REGION Network 3: Vaciado
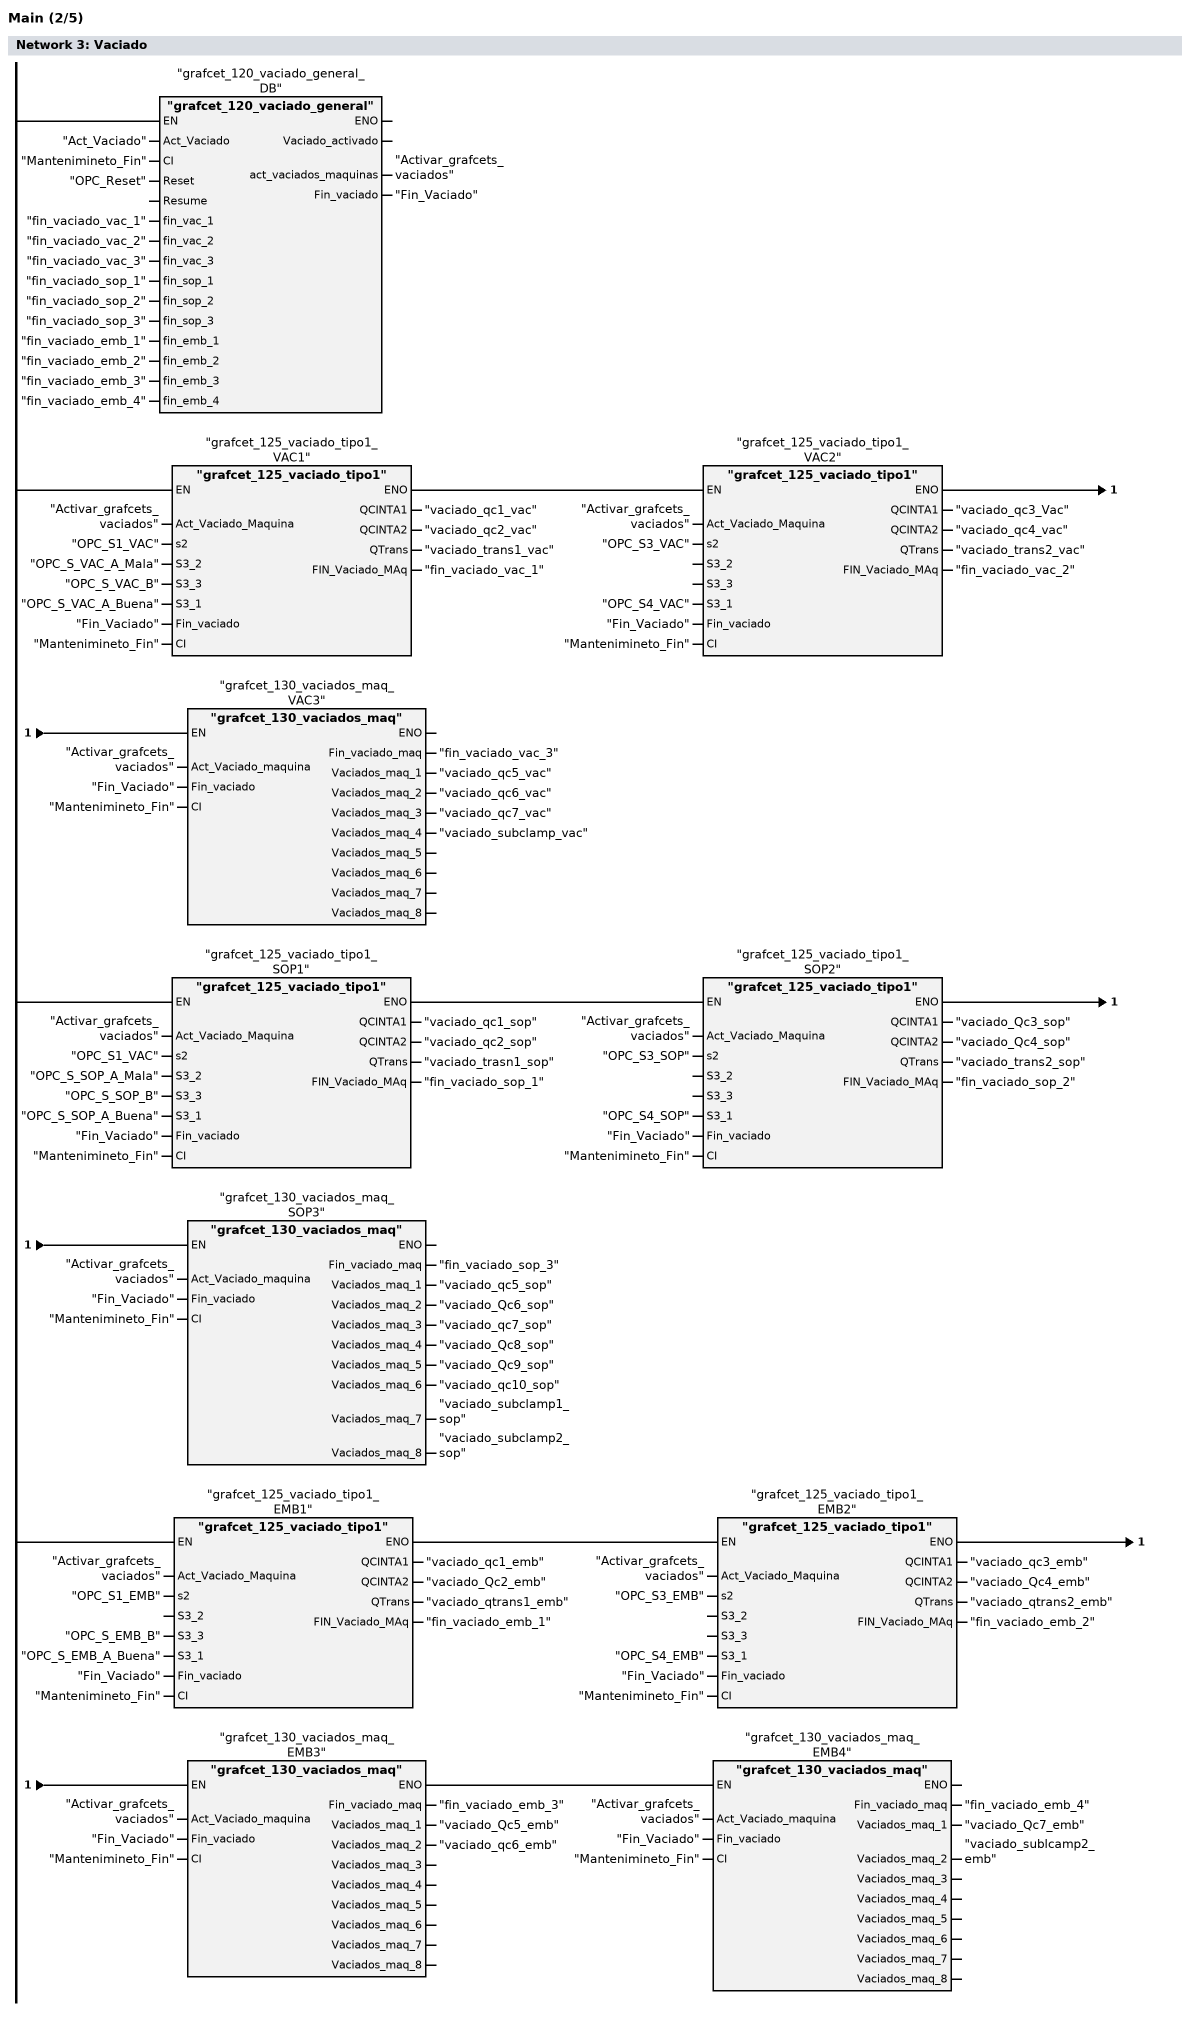
   RUNG wire#powerrail
      "grafcet_120_vaciado_general_DB"(Act_Vaciado := "Act_Vaciado", CI := "Mantenimineto_Fin", Reset := "OPC_Reset", Resume :=, fin_vac_1 := "fin_vaciado_vac_1", fin_vac_2 := "fin_vaciado_vac_2", fin_vac_3 := "fin_vaciado_vac_3", fin_sop_1 := "fin_vaciado_sop_1", fin_sop_2 := "fin_vaciado_sop_2", fin_sop_3 := "fin_vaciado_sop_3", fin_emb_1 := "fin_vaciado_emb_1", fin_emb_2 := "fin_vaciado_emb_2", fin_emb_3 := "fin_vaciado_emb_3", fin_emb_4 := "fin_vaciado_emb_4", Vaciado_activado =>, act_vaciados_maquinas => "Activar_grafcets_vaciados", Fin_vaciado => "Fin_Vaciado")
   END_RUNG
   RUNG wire#powerrail
      "grafcet_125_vaciado_tipo1_VAC1"(Act_Vaciado_Maquina := "Activar_grafcets_vaciados", s2 := "OPC_S1_VAC", S3_2 := "OPC_S_VAC_A_Mala", S3_3 := "OPC_S_VAC_B", S3_1 := "OPC_S_VAC_A_Buena", Fin_vaciado := "Fin_Vaciado", CI := "Mantenimineto_Fin", QCINTA1 => "vaciado_qc1_vac", QCINTA2 => "vaciado_qc2_vac", QTrans => "vaciado_trans1_vac", FIN_Vaciado_MAq => "fin_vaciado_vac_1")
      "grafcet_125_vaciado_tipo1_VAC2"(Act_Vaciado_Maquina := "Activar_grafcets_vaciados", s2 := "OPC_S3_VAC", S3_2 :=, S3_3 :=, S3_1 := "OPC_S4_VAC", Fin_vaciado := "Fin_Vaciado", CI := "Mantenimineto_Fin", QCINTA1 => "vaciado_qc3_Vac", QCINTA2 => "vaciado_qc4_vac", QTrans => "vaciado_trans2_vac", FIN_Vaciado_MAq => "fin_vaciado_vac_2")
      "grafcet_130_vaciados_maq_VAC3"(Act_Vaciado_maquina := "Activar_grafcets_vaciados", Fin_vaciado := "Fin_Vaciado", CI := "Mantenimineto_Fin", Fin_vaciado_maq => "fin_vaciado_vac_3", Vaciados_maq_1 => "vaciado_qc5_vac", Vaciados_maq_2 => "vaciado_qc6_vac", Vaciados_maq_3 => "vaciado_qc7_vac", Vaciados_maq_4 => "vaciado_subclamp_vac", Vaciados_maq_5 =>, Vaciados_maq_6 =>, Vaciados_maq_7 =>, Vaciados_maq_8 =>)
   END_RUNG
   RUNG wire#powerrail
      "grafcet_125_vaciado_tipo1_SOP1"(Act_Vaciado_Maquina := "Activar_grafcets_vaciados", s2 := "OPC_S1_VAC", S3_2 := "OPC_S_SOP_A_Mala", S3_3 := "OPC_S_SOP_B", S3_1 := "OPC_S_SOP_A_Buena", Fin_vaciado := "Fin_Vaciado", CI := "Mantenimineto_Fin", QCINTA1 => "vaciado_qc1_sop", QCINTA2 => "vaciado_qc2_sop", QTrans => "vaciado_trasn1_sop", FIN_Vaciado_MAq => "fin_vaciado_sop_1")
      "grafcet_125_vaciado_tipo1_SOP2"(Act_Vaciado_Maquina := "Activar_grafcets_vaciados", s2 := "OPC_S3_SOP", S3_2 :=, S3_3 :=, S3_1 := "OPC_S4_SOP", Fin_vaciado := "Fin_Vaciado", CI := "Mantenimineto_Fin", QCINTA1 => "vaciado_Qc3_sop", QCINTA2 => "vaciado_Qc4_sop", QTrans => "vaciado_trans2_sop", FIN_Vaciado_MAq => "fin_vaciado_sop_2")
      "grafcet_130_vaciados_maq_SOP3"(Act_Vaciado_maquina := "Activar_grafcets_vaciados", Fin_vaciado := "Fin_Vaciado", CI := "Mantenimineto_Fin", Fin_vaciado_maq => "fin_vaciado_sop_3", Vaciados_maq_1 => "vaciado_qc5_sop", Vaciados_maq_2 => "vaciado_Qc6_sop", Vaciados_maq_3 => "vaciado_qc7_sop", Vaciados_maq_4 => "vaciado_Qc8_sop", Vaciados_maq_5 => "vaciado_Qc9_sop", Vaciados_maq_6 => "vaciado_qc10_sop", Vaciados_maq_7 => "vaciado_subclamp1_sop", Vaciados_maq_8 => "vaciado_subclamp2_sop")
   END_RUNG
   RUNG wire#powerrail
      "grafcet_125_vaciado_tipo1_EMB1"(Act_Vaciado_Maquina := "Activar_grafcets_vaciados", s2 := "OPC_S1_EMB", S3_2 :=, S3_3 := "OPC_S_EMB_B", S3_1 := "OPC_S_EMB_A_Buena", Fin_vaciado := "Fin_Vaciado", CI := "Mantenimineto_Fin", QCINTA1 => "vaciado_qc1_emb", QCINTA2 => "vaciado_Qc2_emb", QTrans => "vaciado_qtrans1_emb", FIN_Vaciado_MAq => "fin_vaciado_emb_1")
      "grafcet_125_vaciado_tipo1_EMB2"(Act_Vaciado_Maquina := "Activar_grafcets_vaciados", s2 := "OPC_S3_EMB", S3_2 :=, S3_3 :=, S3_1 := "OPC_S4_EMB", Fin_vaciado := "Fin_Vaciado", CI := "Mantenimineto_Fin", QCINTA1 => "vaciado_qc3_emb", QCINTA2 => "vaciado_Qc4_emb", QTrans => "vaciado_qtrans2_emb", FIN_Vaciado_MAq => "fin_vaciado_emb_2")
      "grafcet_130_vaciados_maq_EMB3"(Act_Vaciado_maquina := "Activar_grafcets_vaciados", Fin_vaciado := "Fin_Vaciado", CI := "Mantenimineto_Fin", Fin_vaciado_maq => "fin_vaciado_emb_3", Vaciados_maq_1 => "vaciado_Qc5_emb", Vaciados_maq_2 => "vaciado_qc6_emb", Vaciados_maq_3 =>, Vaciados_maq_4 =>, Vaciados_maq_5 =>, Vaciados_maq_6 =>, Vaciados_maq_7 =>, Vaciados_maq_8 =>)
      "grafcet_130_vaciados_maq_EMB4"(Act_Vaciado_maquina := "Activar_grafcets_vaciados", Fin_vaciado := "Fin_Vaciado", CI := "Mantenimineto_Fin", Fin_vaciado_maq => "fin_vaciado_emb_4", Vaciados_maq_1 => "vaciado_Qc7_emb", Vaciados_maq_2 => "vaciado_sublcamp2_emb", Vaciados_maq_3 =>, Vaciados_maq_4 =>, Vaciados_maq_5 =>, Vaciados_maq_6 =>, Vaciados_maq_7 =>, Vaciados_maq_8 =>)
   END_RUNG
   // the same network as SCL:
   "grafcet_120_vaciado_general_DB"(Act_Vaciado := "Act_Vaciado",   // "grafcet_120_vaciado_general"
                           CI := "Mantenimineto_Fin",
                           Reset := "OPC_Reset",
                           fin_vac_1 := "fin_vaciado_vac_1",
                           fin_vac_2 := "fin_vaciado_vac_2",
                           fin_vac_3 := "fin_vaciado_vac_3",
                           fin_sop_1 := "fin_vaciado_sop_1",
                           fin_sop_2 := "fin_vaciado_sop_2",
                           fin_sop_3 := "fin_vaciado_sop_3",
                           fin_emb_1 := "fin_vaciado_emb_1",
                           fin_emb_2 := "fin_vaciado_emb_2",
                           fin_emb_3 := "fin_vaciado_emb_3",
                           fin_emb_4 := "fin_vaciado_emb_4",
                           act_vaciados_maquinas => "Activar_grafcets_vaciados",
                           Fin_vaciado => "Fin_Vaciado");
   "grafcet_125_vaciado_tipo1_VAC1"(Act_Vaciado_Maquina := "Activar_grafcets_vaciados",   // "grafcet_125_vaciado_tipo1"
                           s2 := "OPC_S1_VAC",
                           S3_2 := "OPC_S_VAC_A_Mala",
                           S3_3 := "OPC_S_VAC_B",
                           S3_1 := "OPC_S_VAC_A_Buena",
                           Fin_vaciado := "Fin_Vaciado",
                           CI := "Mantenimineto_Fin",
                           QCINTA1 => "vaciado_qc1_vac",
                           QCINTA2 => "vaciado_qc2_vac",
                           QTrans => "vaciado_trans1_vac",
                           FIN_Vaciado_MAq => "fin_vaciado_vac_1",
                           ENO => #_w1);
   "grafcet_125_vaciado_tipo1_VAC2"(EN := #_w1,   // "grafcet_125_vaciado_tipo1"
                           Act_Vaciado_Maquina := "Activar_grafcets_vaciados",
                           s2 := "OPC_S3_VAC",
                           S3_1 := "OPC_S4_VAC",
                           Fin_vaciado := "Fin_Vaciado",
                           CI := "Mantenimineto_Fin",
                           QCINTA1 => "vaciado_qc3_Vac",
                           QCINTA2 => "vaciado_qc4_vac",
                           QTrans => "vaciado_trans2_vac",
                           FIN_Vaciado_MAq => "fin_vaciado_vac_2",
                           ENO => #_w2);
   IF #_w2 THEN
       "grafcet_130_vaciados_maq_VAC3"(Act_Vaciado_maquina := "Activar_grafcets_vaciados",   // "grafcet_130_vaciados_maq"
                               Fin_vaciado := "Fin_Vaciado",
                               CI := "Mantenimineto_Fin",
                               Fin_vaciado_maq => "fin_vaciado_vac_3",
                               Vaciados_maq_1 => "vaciado_qc5_vac",
                               Vaciados_maq_2 => "vaciado_qc6_vac",
                               Vaciados_maq_3 => "vaciado_qc7_vac",
                               Vaciados_maq_4 => "vaciado_subclamp_vac");
   END_IF;
   "grafcet_125_vaciado_tipo1_SOP1"(Act_Vaciado_Maquina := "Activar_grafcets_vaciados",   // "grafcet_125_vaciado_tipo1"
                           s2 := "OPC_S1_VAC",
                           S3_2 := "OPC_S_SOP_A_Mala",
                           S3_3 := "OPC_S_SOP_B",
                           S3_1 := "OPC_S_SOP_A_Buena",
                           Fin_vaciado := "Fin_Vaciado",
                           CI := "Mantenimineto_Fin",
                           QCINTA1 => "vaciado_qc1_sop",
                           QCINTA2 => "vaciado_qc2_sop",
                           QTrans => "vaciado_trasn1_sop",
                           FIN_Vaciado_MAq => "fin_vaciado_sop_1",
                           ENO => #_w3);
   "grafcet_125_vaciado_tipo1_SOP2"(EN := #_w3,   // "grafcet_125_vaciado_tipo1"
                           Act_Vaciado_Maquina := "Activar_grafcets_vaciados",
                           s2 := "OPC_S3_SOP",
                           S3_1 := "OPC_S4_SOP",
                           Fin_vaciado := "Fin_Vaciado",
                           CI := "Mantenimineto_Fin",
                           QCINTA1 => "vaciado_Qc3_sop",
                           QCINTA2 => "vaciado_Qc4_sop",
                           QTrans => "vaciado_trans2_sop",
                           FIN_Vaciado_MAq => "fin_vaciado_sop_2",
                           ENO => #_w4);
   IF #_w4 THEN
       "grafcet_130_vaciados_maq_SOP3"(Act_Vaciado_maquina := "Activar_grafcets_vaciados",   // "grafcet_130_vaciados_maq"
                               Fin_vaciado := "Fin_Vaciado",
                               CI := "Mantenimineto_Fin",
                               Fin_vaciado_maq => "fin_vaciado_sop_3",
                               Vaciados_maq_1 => "vaciado_qc5_sop",
                               Vaciados_maq_2 => "vaciado_Qc6_sop",
                               Vaciados_maq_3 => "vaciado_qc7_sop",
                               Vaciados_maq_4 => "vaciado_Qc8_sop",
                               Vaciados_maq_5 => "vaciado_Qc9_sop",
                               Vaciados_maq_6 => "vaciado_qc10_sop",
                               Vaciados_maq_7 => "vaciado_subclamp1_sop",
                               Vaciados_maq_8 => "vaciado_subclamp2_sop");
   END_IF;
   "grafcet_125_vaciado_tipo1_EMB1"(Act_Vaciado_Maquina := "Activar_grafcets_vaciados",   // "grafcet_125_vaciado_tipo1"
                           s2 := "OPC_S1_EMB",
                           S3_3 := "OPC_S_EMB_B",
                           S3_1 := "OPC_S_EMB_A_Buena",
                           Fin_vaciado := "Fin_Vaciado",
                           CI := "Mantenimineto_Fin",
                           QCINTA1 => "vaciado_qc1_emb",
                           QCINTA2 => "vaciado_Qc2_emb",
                           QTrans => "vaciado_qtrans1_emb",
                           FIN_Vaciado_MAq => "fin_vaciado_emb_1",
                           ENO => #_w5);
   "grafcet_125_vaciado_tipo1_EMB2"(EN := #_w5,   // "grafcet_125_vaciado_tipo1"
                           Act_Vaciado_Maquina := "Activar_grafcets_vaciados",
                           s2 := "OPC_S3_EMB",
                           S3_1 := "OPC_S4_EMB",
                           Fin_vaciado := "Fin_Vaciado",
                           CI := "Mantenimineto_Fin",
                           QCINTA1 => "vaciado_qc3_emb",
                           QCINTA2 => "vaciado_Qc4_emb",
                           QTrans => "vaciado_qtrans2_emb",
                           FIN_Vaciado_MAq => "fin_vaciado_emb_2",
                           ENO => #_w6);
   "grafcet_130_vaciados_maq_EMB3"(EN := #_w6,   // "grafcet_130_vaciados_maq"
                           Act_Vaciado_maquina := "Activar_grafcets_vaciados",
                           Fin_vaciado := "Fin_Vaciado",
                           CI := "Mantenimineto_Fin",
                           Fin_vaciado_maq => "fin_vaciado_emb_3",
                           Vaciados_maq_1 => "vaciado_Qc5_emb",
                           Vaciados_maq_2 => "vaciado_qc6_emb",
                           ENO => #_w7);
   IF #_w7 THEN
       "grafcet_130_vaciados_maq_EMB4"(Act_Vaciado_maquina := "Activar_grafcets_vaciados",   // "grafcet_130_vaciados_maq"
                               Fin_vaciado := "Fin_Vaciado",
                               CI := "Mantenimineto_Fin",
                               Fin_vaciado_maq => "fin_vaciado_emb_4",
                               Vaciados_maq_1 => "vaciado_Qc7_emb",
                               Vaciados_maq_2 => "vaciado_sublcamp2_emb");
   END_IF;
END_REGION

REGION Network 4: Maquina Vacunas
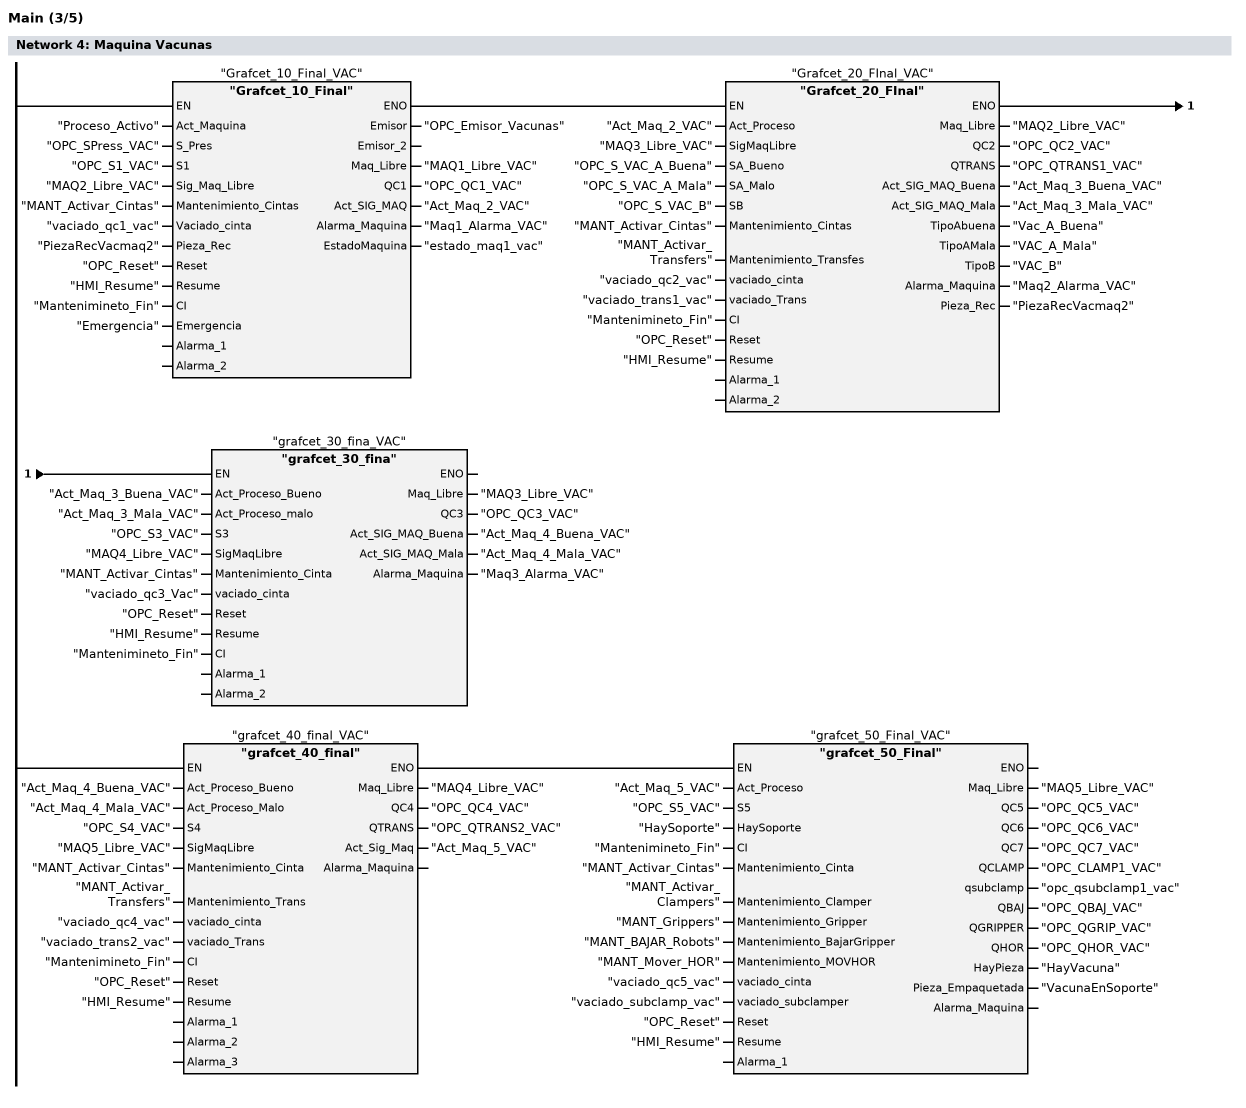
   RUNG wire#powerrail
      "Grafcet_10_Final_VAC"(Act_Maquina := "Proceso_Activo", S_Pres := "OPC_SPress_VAC", S1 := "OPC_S1_VAC", Sig_Maq_Libre := "MAQ2_Libre_VAC", Mantenimiento_Cintas := "MANT_Activar_Cintas", Vaciado_cinta := "vaciado_qc1_vac", Pieza_Rec := "PiezaRecVacmaq2", Reset := "OPC_Reset", Resume := "HMI_Resume", CI := "Mantenimineto_Fin", Emergencia := "Emergencia", Alarma_1 :=, Alarma_2 :=, Emisor => "OPC_Emisor_Vacunas", Emisor_2 =>, Maq_Libre => "MAQ1_Libre_VAC", QC1 => "OPC_QC1_VAC", Act_SIG_MAQ => "Act_Maq_2_VAC", Alarma_Maquina => "Maq1_Alarma_VAC", EstadoMaquina => "estado_maq1_vac")
      "Grafcet_20_FInal_VAC"(Act_Proceso := "Act_Maq_2_VAC", SigMaqLibre := "MAQ3_Libre_VAC", SA_Bueno := "OPC_S_VAC_A_Buena", SA_Malo := "OPC_S_VAC_A_Mala", SB := "OPC_S_VAC_B", Mantenimiento_Cintas := "MANT_Activar_Cintas", Mantenimiento_Transfes := "MANT_Activar_Transfers", vaciado_cinta := "vaciado_qc2_vac", vaciado_Trans := "vaciado_trans1_vac", CI := "Mantenimineto_Fin", Reset := "OPC_Reset", Resume := "HMI_Resume", Alarma_1 :=, Alarma_2 :=, Maq_Libre => "MAQ2_Libre_VAC", QC2 => "OPC_QC2_VAC", QTRANS => "OPC_QTRANS1_VAC", Act_SIG_MAQ_Buena => "Act_Maq_3_Buena_VAC", Act_SIG_MAQ_Mala => "Act_Maq_3_Mala_VAC", TipoAbuena => "Vac_A_Buena", TipoAMala => "VAC_A_Mala", TipoB => "VAC_B", Alarma_Maquina => "Maq2_Alarma_VAC", Pieza_Rec => "PiezaRecVacmaq2")
      "grafcet_30_fina_VAC"(Act_Proceso_Bueno := "Act_Maq_3_Buena_VAC", Act_Proceso_malo := "Act_Maq_3_Mala_VAC", S3 := "OPC_S3_VAC", SigMaqLibre := "MAQ4_Libre_VAC", Mantenimiento_Cinta := "MANT_Activar_Cintas", vaciado_cinta := "vaciado_qc3_Vac", Reset := "OPC_Reset", Resume := "HMI_Resume", CI := "Mantenimineto_Fin", Alarma_1 :=, Alarma_2 :=, Maq_Libre => "MAQ3_Libre_VAC", QC3 => "OPC_QC3_VAC", Act_SIG_MAQ_Buena => "Act_Maq_4_Buena_VAC", Act_SIG_MAQ_Mala => "Act_Maq_4_Mala_VAC", Alarma_Maquina => "Maq3_Alarma_VAC")
   END_RUNG
   RUNG wire#powerrail
      "grafcet_40_final_VAC"(Act_Proceso_Bueno := "Act_Maq_4_Buena_VAC", Act_Proceso_Malo := "Act_Maq_4_Mala_VAC", S4 := "OPC_S4_VAC", SigMaqLibre := "MAQ5_Libre_VAC", Mantenimiento_Cinta := "MANT_Activar_Cintas", Mantenimiento_Trans := "MANT_Activar_Transfers", vaciado_cinta := "vaciado_qc4_vac", vaciado_Trans := "vaciado_trans2_vac", CI := "Mantenimineto_Fin", Reset := "OPC_Reset", Resume := "HMI_Resume", Alarma_1 :=, Alarma_2 :=, Alarma_3 :=, Maq_Libre => "MAQ4_Libre_VAC", QC4 => "OPC_QC4_VAC", QTRANS => "OPC_QTRANS2_VAC", Act_Sig_Maq => "Act_Maq_5_VAC", Alarma_Maquina =>)
      "grafcet_50_Final_VAC"(Act_Proceso := "Act_Maq_5_VAC", S5 := "OPC_S5_VAC", HaySoporte := "HaySoporte", CI := "Mantenimineto_Fin", Mantenimiento_Cinta := "MANT_Activar_Cintas", Mantenimiento_Clamper := "MANT_Activar_Clampers", Mantenimiento_Gripper := "MANT_Grippers", Mantenimiento_BajarGripper := "MANT_BAJAR_Robots", Mantenimiento_MOVHOR := "MANT_Mover_HOR", vaciado_cinta := "vaciado_qc5_vac", vaciado_subclamper := "vaciado_subclamp_vac", Reset := "OPC_Reset", Resume := "HMI_Resume", Alarma_1 :=, Maq_Libre => "MAQ5_Libre_VAC", QC5 => "OPC_QC5_VAC", QC6 => "OPC_QC6_VAC", QC7 => "OPC_QC7_VAC", QCLAMP => "OPC_CLAMP1_VAC", qsubclamp => "opc_qsubclamp1_vac", QBAJ => "OPC_QBAJ_VAC", QGRIPPER => "OPC_QGRIP_VAC", QHOR => "OPC_QHOR_VAC", HayPieza => "HayVacuna", Pieza_Empaquetada => "VacunaEnSoporte", Alarma_Maquina =>)
   END_RUNG
   // the same network as SCL:
   "Grafcet_10_Final_VAC"(Act_Maquina := "Proceso_Activo",   // "Grafcet_10_Final"
                          S_Pres := "OPC_SPress_VAC",
                          S1 := "OPC_S1_VAC",
                          Sig_Maq_Libre := "MAQ2_Libre_VAC",
                          Mantenimiento_Cintas := "MANT_Activar_Cintas",
                          Vaciado_cinta := "vaciado_qc1_vac",
                          Pieza_Rec := "PiezaRecVacmaq2",
                          Reset := "OPC_Reset",
                          Resume := "HMI_Resume",
                          CI := "Mantenimineto_Fin",
                          Emergencia := "Emergencia",
                          Emisor => "OPC_Emisor_Vacunas",
                          Maq_Libre => "MAQ1_Libre_VAC",
                          QC1 => "OPC_QC1_VAC",
                          Act_SIG_MAQ => "Act_Maq_2_VAC",
                          Alarma_Maquina => "Maq1_Alarma_VAC",
                          EstadoMaquina => "estado_maq1_vac",
                          ENO => #_w1);
   "Grafcet_20_FInal_VAC"(EN := #_w1,   // "Grafcet_20_FInal"
                          Act_Proceso := "Act_Maq_2_VAC",
                          SigMaqLibre := "MAQ3_Libre_VAC",
                          SA_Bueno := "OPC_S_VAC_A_Buena",
                          SA_Malo := "OPC_S_VAC_A_Mala",
                          SB := "OPC_S_VAC_B",
                          Mantenimiento_Cintas := "MANT_Activar_Cintas",
                          Mantenimiento_Transfes := "MANT_Activar_Transfers",
                          vaciado_cinta := "vaciado_qc2_vac",
                          vaciado_Trans := "vaciado_trans1_vac",
                          CI := "Mantenimineto_Fin",
                          Reset := "OPC_Reset",
                          Resume := "HMI_Resume",
                          Maq_Libre => "MAQ2_Libre_VAC",
                          QC2 => "OPC_QC2_VAC",
                          QTRANS => "OPC_QTRANS1_VAC",
                          Act_SIG_MAQ_Buena => "Act_Maq_3_Buena_VAC",
                          Act_SIG_MAQ_Mala => "Act_Maq_3_Mala_VAC",
                          TipoAbuena => "Vac_A_Buena",
                          TipoAMala => "VAC_A_Mala",
                          TipoB => "VAC_B",
                          Alarma_Maquina => "Maq2_Alarma_VAC",
                          Pieza_Rec => "PiezaRecVacmaq2",
                          ENO => #_w2);
   IF #_w2 THEN
       "grafcet_30_fina_VAC"(Act_Proceso_Bueno := "Act_Maq_3_Buena_VAC",   // "grafcet_30_fina"
                             Act_Proceso_malo := "Act_Maq_3_Mala_VAC",
                             S3 := "OPC_S3_VAC",
                             SigMaqLibre := "MAQ4_Libre_VAC",
                             Mantenimiento_Cinta := "MANT_Activar_Cintas",
                             vaciado_cinta := "vaciado_qc3_Vac",
                             Reset := "OPC_Reset",
                             Resume := "HMI_Resume",
                             CI := "Mantenimineto_Fin",
                             Maq_Libre => "MAQ3_Libre_VAC",
                             QC3 => "OPC_QC3_VAC",
                             Act_SIG_MAQ_Buena => "Act_Maq_4_Buena_VAC",
                             Act_SIG_MAQ_Mala => "Act_Maq_4_Mala_VAC",
                             Alarma_Maquina => "Maq3_Alarma_VAC");
   END_IF;
   "grafcet_40_final_VAC"(Act_Proceso_Bueno := "Act_Maq_4_Buena_VAC",   // "grafcet_40_final"
                          Act_Proceso_Malo := "Act_Maq_4_Mala_VAC",
                          S4 := "OPC_S4_VAC",
                          SigMaqLibre := "MAQ5_Libre_VAC",
                          Mantenimiento_Cinta := "MANT_Activar_Cintas",
                          Mantenimiento_Trans := "MANT_Activar_Transfers",
                          vaciado_cinta := "vaciado_qc4_vac",
                          vaciado_Trans := "vaciado_trans2_vac",
                          CI := "Mantenimineto_Fin",
                          Reset := "OPC_Reset",
                          Resume := "HMI_Resume",
                          Maq_Libre => "MAQ4_Libre_VAC",
                          QC4 => "OPC_QC4_VAC",
                          QTRANS => "OPC_QTRANS2_VAC",
                          Act_Sig_Maq => "Act_Maq_5_VAC",
                          ENO => #_w3);
   IF #_w3 THEN
       "grafcet_50_Final_VAC"(Act_Proceso := "Act_Maq_5_VAC",   // "grafcet_50_Final"
                              S5 := "OPC_S5_VAC",
                              HaySoporte := "HaySoporte",
                              CI := "Mantenimineto_Fin",
                              Mantenimiento_Cinta := "MANT_Activar_Cintas",
                              Mantenimiento_Clamper := "MANT_Activar_Clampers",
                              Mantenimiento_Gripper := "MANT_Grippers",
                              Mantenimiento_BajarGripper := "MANT_BAJAR_Robots",
                              Mantenimiento_MOVHOR := "MANT_Mover_HOR",
                              vaciado_cinta := "vaciado_qc5_vac",
                              vaciado_subclamper := "vaciado_subclamp_vac",
                              Reset := "OPC_Reset",
                              Resume := "HMI_Resume",
                              Maq_Libre => "MAQ5_Libre_VAC",
                              QC5 => "OPC_QC5_VAC",
                              QC6 => "OPC_QC6_VAC",
                              QC7 => "OPC_QC7_VAC",
                              QCLAMP => "OPC_CLAMP1_VAC",
                              qsubclamp => "opc_qsubclamp1_vac",
                              QBAJ => "OPC_QBAJ_VAC",
                              QGRIPPER => "OPC_QGRIP_VAC",
                              QHOR => "OPC_QHOR_VAC",
                              HayPieza => "HayVacuna",
                              Pieza_Empaquetada => "VacunaEnSoporte");
   END_IF;
END_REGION

REGION Network 5: Maquina Soporte
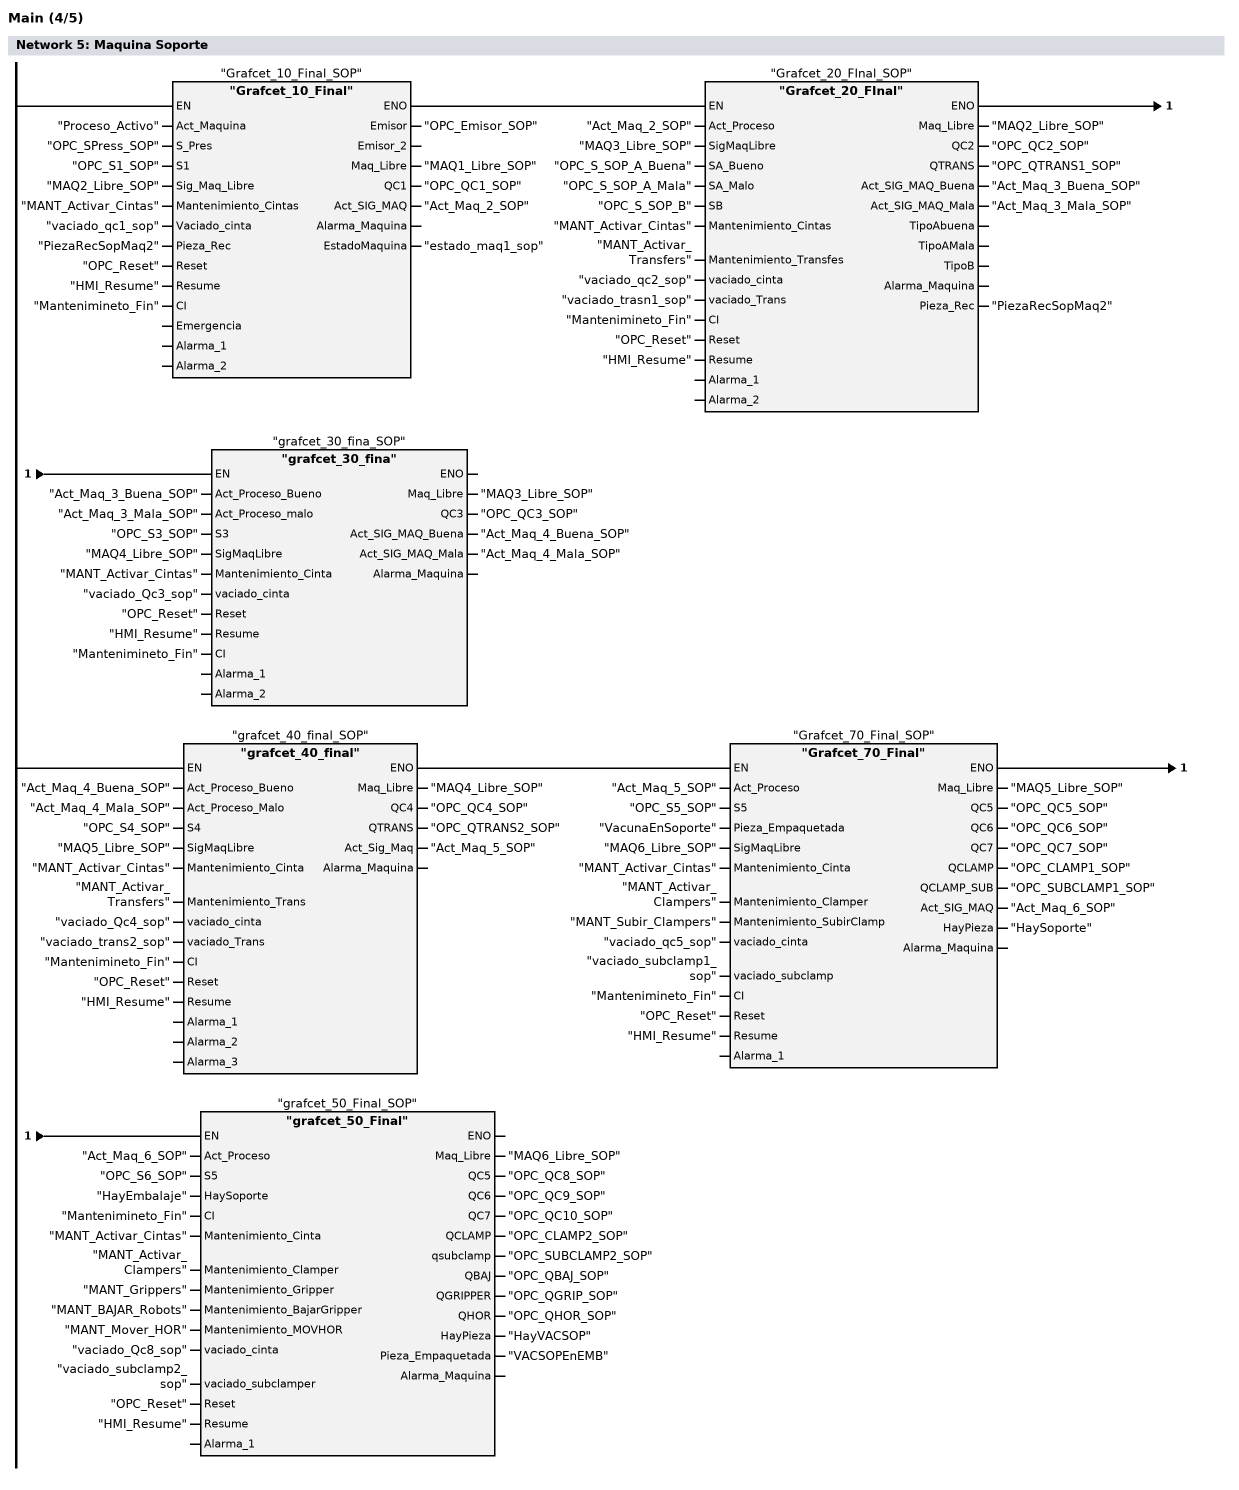
   RUNG wire#powerrail
      "Grafcet_10_Final_SOP"(Act_Maquina := "Proceso_Activo", S_Pres := "OPC_SPress_SOP", S1 := "OPC_S1_SOP", Sig_Maq_Libre := "MAQ2_Libre_SOP", Mantenimiento_Cintas := "MANT_Activar_Cintas", Vaciado_cinta := "vaciado_qc1_sop", Pieza_Rec := "PiezaRecSopMaq2", Reset := "OPC_Reset", Resume := "HMI_Resume", CI := "Mantenimineto_Fin", Emergencia :=, Alarma_1 :=, Alarma_2 :=, Emisor => "OPC_Emisor_SOP", Emisor_2 =>, Maq_Libre => "MAQ1_Libre_SOP", QC1 => "OPC_QC1_SOP", Act_SIG_MAQ => "Act_Maq_2_SOP", Alarma_Maquina =>, EstadoMaquina => "estado_maq1_sop")
      "Grafcet_20_FInal_SOP"(Act_Proceso := "Act_Maq_2_SOP", SigMaqLibre := "MAQ3_Libre_SOP", SA_Bueno := "OPC_S_SOP_A_Buena", SA_Malo := "OPC_S_SOP_A_Mala", SB := "OPC_S_SOP_B", Mantenimiento_Cintas := "MANT_Activar_Cintas", Mantenimiento_Transfes := "MANT_Activar_Transfers", vaciado_cinta := "vaciado_qc2_sop", vaciado_Trans := "vaciado_trasn1_sop", CI := "Mantenimineto_Fin", Reset := "OPC_Reset", Resume := "HMI_Resume", Alarma_1 :=, Alarma_2 :=, Maq_Libre => "MAQ2_Libre_SOP", QC2 => "OPC_QC2_SOP", QTRANS => "OPC_QTRANS1_SOP", Act_SIG_MAQ_Buena => "Act_Maq_3_Buena_SOP", Act_SIG_MAQ_Mala => "Act_Maq_3_Mala_SOP", TipoAbuena =>, TipoAMala =>, TipoB =>, Alarma_Maquina =>, Pieza_Rec => "PiezaRecSopMaq2")
      "grafcet_30_fina_SOP"(Act_Proceso_Bueno := "Act_Maq_3_Buena_SOP", Act_Proceso_malo := "Act_Maq_3_Mala_SOP", S3 := "OPC_S3_SOP", SigMaqLibre := "MAQ4_Libre_SOP", Mantenimiento_Cinta := "MANT_Activar_Cintas", vaciado_cinta := "vaciado_Qc3_sop", Reset := "OPC_Reset", Resume := "HMI_Resume", CI := "Mantenimineto_Fin", Alarma_1 :=, Alarma_2 :=, Maq_Libre => "MAQ3_Libre_SOP", QC3 => "OPC_QC3_SOP", Act_SIG_MAQ_Buena => "Act_Maq_4_Buena_SOP", Act_SIG_MAQ_Mala => "Act_Maq_4_Mala_SOP", Alarma_Maquina =>)
   END_RUNG
   RUNG wire#powerrail
      "grafcet_40_final_SOP"(Act_Proceso_Bueno := "Act_Maq_4_Buena_SOP", Act_Proceso_Malo := "Act_Maq_4_Mala_SOP", S4 := "OPC_S4_SOP", SigMaqLibre := "MAQ5_Libre_SOP", Mantenimiento_Cinta := "MANT_Activar_Cintas", Mantenimiento_Trans := "MANT_Activar_Transfers", vaciado_cinta := "vaciado_Qc4_sop", vaciado_Trans := "vaciado_trans2_sop", CI := "Mantenimineto_Fin", Reset := "OPC_Reset", Resume := "HMI_Resume", Alarma_1 :=, Alarma_2 :=, Alarma_3 :=, Maq_Libre => "MAQ4_Libre_SOP", QC4 => "OPC_QC4_SOP", QTRANS => "OPC_QTRANS2_SOP", Act_Sig_Maq => "Act_Maq_5_SOP", Alarma_Maquina =>)
      "Grafcet_70_Final_SOP"(Act_Proceso := "Act_Maq_5_SOP", S5 := "OPC_S5_SOP", Pieza_Empaquetada := "VacunaEnSoporte", SigMaqLibre := "MAQ6_Libre_SOP", Mantenimiento_Cinta := "MANT_Activar_Cintas", Mantenimiento_Clamper := "MANT_Activar_Clampers", Mantenimiento_SubirClamp := "MANT_Subir_Clampers", vaciado_cinta := "vaciado_qc5_sop", vaciado_subclamp := "vaciado_subclamp1_sop", CI := "Mantenimineto_Fin", Reset := "OPC_Reset", Resume := "HMI_Resume", Alarma_1 :=, Maq_Libre => "MAQ5_Libre_SOP", QC5 => "OPC_QC5_SOP", QC6 => "OPC_QC6_SOP", QC7 => "OPC_QC7_SOP", QCLAMP => "OPC_CLAMP1_SOP", QCLAMP_SUB => "OPC_SUBCLAMP1_SOP", Act_SIG_MAQ => "Act_Maq_6_SOP", HayPieza => "HaySoporte", Alarma_Maquina =>)
      "grafcet_50_Final_SOP"(Act_Proceso := "Act_Maq_6_SOP", S5 := "OPC_S6_SOP", HaySoporte := "HayEmbalaje", CI := "Mantenimineto_Fin", Mantenimiento_Cinta := "MANT_Activar_Cintas", Mantenimiento_Clamper := "MANT_Activar_Clampers", Mantenimiento_Gripper := "MANT_Grippers", Mantenimiento_BajarGripper := "MANT_BAJAR_Robots", Mantenimiento_MOVHOR := "MANT_Mover_HOR", vaciado_cinta := "vaciado_Qc8_sop", vaciado_subclamper := "vaciado_subclamp2_sop", Reset := "OPC_Reset", Resume := "HMI_Resume", Alarma_1 :=, Maq_Libre => "MAQ6_Libre_SOP", QC5 => "OPC_QC8_SOP", QC6 => "OPC_QC9_SOP", QC7 => "OPC_QC10_SOP", QCLAMP => "OPC_CLAMP2_SOP", qsubclamp => "OPC_SUBCLAMP2_SOP", QBAJ => "OPC_QBAJ_SOP", QGRIPPER => "OPC_QGRIP_SOP", QHOR => "OPC_QHOR_SOP", HayPieza => "HayVACSOP", Pieza_Empaquetada => "VACSOPEnEMB", Alarma_Maquina =>)
   END_RUNG
   // the same network as SCL:
   "Grafcet_10_Final_SOP"(Act_Maquina := "Proceso_Activo",   // "Grafcet_10_Final"
                          S_Pres := "OPC_SPress_SOP",
                          S1 := "OPC_S1_SOP",
                          Sig_Maq_Libre := "MAQ2_Libre_SOP",
                          Mantenimiento_Cintas := "MANT_Activar_Cintas",
                          Vaciado_cinta := "vaciado_qc1_sop",
                          Pieza_Rec := "PiezaRecSopMaq2",
                          Reset := "OPC_Reset",
                          Resume := "HMI_Resume",
                          CI := "Mantenimineto_Fin",
                          Emisor => "OPC_Emisor_SOP",
                          Maq_Libre => "MAQ1_Libre_SOP",
                          QC1 => "OPC_QC1_SOP",
                          Act_SIG_MAQ => "Act_Maq_2_SOP",
                          EstadoMaquina => "estado_maq1_sop",
                          ENO => #_w1);
   "Grafcet_20_FInal_SOP"(EN := #_w1,   // "Grafcet_20_FInal"
                          Act_Proceso := "Act_Maq_2_SOP",
                          SigMaqLibre := "MAQ3_Libre_SOP",
                          SA_Bueno := "OPC_S_SOP_A_Buena",
                          SA_Malo := "OPC_S_SOP_A_Mala",
                          SB := "OPC_S_SOP_B",
                          Mantenimiento_Cintas := "MANT_Activar_Cintas",
                          Mantenimiento_Transfes := "MANT_Activar_Transfers",
                          vaciado_cinta := "vaciado_qc2_sop",
                          vaciado_Trans := "vaciado_trasn1_sop",
                          CI := "Mantenimineto_Fin",
                          Reset := "OPC_Reset",
                          Resume := "HMI_Resume",
                          Maq_Libre => "MAQ2_Libre_SOP",
                          QC2 => "OPC_QC2_SOP",
                          QTRANS => "OPC_QTRANS1_SOP",
                          Act_SIG_MAQ_Buena => "Act_Maq_3_Buena_SOP",
                          Act_SIG_MAQ_Mala => "Act_Maq_3_Mala_SOP",
                          Pieza_Rec => "PiezaRecSopMaq2",
                          ENO => #_w2);
   IF #_w2 THEN
       "grafcet_30_fina_SOP"(Act_Proceso_Bueno := "Act_Maq_3_Buena_SOP",   // "grafcet_30_fina"
                             Act_Proceso_malo := "Act_Maq_3_Mala_SOP",
                             S3 := "OPC_S3_SOP",
                             SigMaqLibre := "MAQ4_Libre_SOP",
                             Mantenimiento_Cinta := "MANT_Activar_Cintas",
                             vaciado_cinta := "vaciado_Qc3_sop",
                             Reset := "OPC_Reset",
                             Resume := "HMI_Resume",
                             CI := "Mantenimineto_Fin",
                             Maq_Libre => "MAQ3_Libre_SOP",
                             QC3 => "OPC_QC3_SOP",
                             Act_SIG_MAQ_Buena => "Act_Maq_4_Buena_SOP",
                             Act_SIG_MAQ_Mala => "Act_Maq_4_Mala_SOP");
   END_IF;
   "grafcet_40_final_SOP"(Act_Proceso_Bueno := "Act_Maq_4_Buena_SOP",   // "grafcet_40_final"
                          Act_Proceso_Malo := "Act_Maq_4_Mala_SOP",
                          S4 := "OPC_S4_SOP",
                          SigMaqLibre := "MAQ5_Libre_SOP",
                          Mantenimiento_Cinta := "MANT_Activar_Cintas",
                          Mantenimiento_Trans := "MANT_Activar_Transfers",
                          vaciado_cinta := "vaciado_Qc4_sop",
                          vaciado_Trans := "vaciado_trans2_sop",
                          CI := "Mantenimineto_Fin",
                          Reset := "OPC_Reset",
                          Resume := "HMI_Resume",
                          Maq_Libre => "MAQ4_Libre_SOP",
                          QC4 => "OPC_QC4_SOP",
                          QTRANS => "OPC_QTRANS2_SOP",
                          Act_Sig_Maq => "Act_Maq_5_SOP",
                          ENO => #_w3);
   "Grafcet_70_Final_SOP"(EN := #_w3,   // "Grafcet_70_Final"
                          Act_Proceso := "Act_Maq_5_SOP",
                          S5 := "OPC_S5_SOP",
                          Pieza_Empaquetada := "VacunaEnSoporte",
                          SigMaqLibre := "MAQ6_Libre_SOP",
                          Mantenimiento_Cinta := "MANT_Activar_Cintas",
                          Mantenimiento_Clamper := "MANT_Activar_Clampers",
                          Mantenimiento_SubirClamp := "MANT_Subir_Clampers",
                          vaciado_cinta := "vaciado_qc5_sop",
                          vaciado_subclamp := "vaciado_subclamp1_sop",
                          CI := "Mantenimineto_Fin",
                          Reset := "OPC_Reset",
                          Resume := "HMI_Resume",
                          Maq_Libre => "MAQ5_Libre_SOP",
                          QC5 => "OPC_QC5_SOP",
                          QC6 => "OPC_QC6_SOP",
                          QC7 => "OPC_QC7_SOP",
                          QCLAMP => "OPC_CLAMP1_SOP",
                          QCLAMP_SUB => "OPC_SUBCLAMP1_SOP",
                          Act_SIG_MAQ => "Act_Maq_6_SOP",
                          HayPieza => "HaySoporte",
                          ENO => #_w4);
   IF #_w4 THEN
       "grafcet_50_Final_SOP"(Act_Proceso := "Act_Maq_6_SOP",   // "grafcet_50_Final"
                              S5 := "OPC_S6_SOP",
                              HaySoporte := "HayEmbalaje",
                              CI := "Mantenimineto_Fin",
                              Mantenimiento_Cinta := "MANT_Activar_Cintas",
                              Mantenimiento_Clamper := "MANT_Activar_Clampers",
                              Mantenimiento_Gripper := "MANT_Grippers",
                              Mantenimiento_BajarGripper := "MANT_BAJAR_Robots",
                              Mantenimiento_MOVHOR := "MANT_Mover_HOR",
                              vaciado_cinta := "vaciado_Qc8_sop",
                              vaciado_subclamper := "vaciado_subclamp2_sop",
                              Reset := "OPC_Reset",
                              Resume := "HMI_Resume",
                              Maq_Libre => "MAQ6_Libre_SOP",
                              QC5 => "OPC_QC8_SOP",
                              QC6 => "OPC_QC9_SOP",
                              QC7 => "OPC_QC10_SOP",
                              QCLAMP => "OPC_CLAMP2_SOP",
                              qsubclamp => "OPC_SUBCLAMP2_SOP",
                              QBAJ => "OPC_QBAJ_SOP",
                              QGRIPPER => "OPC_QGRIP_SOP",
                              QHOR => "OPC_QHOR_SOP",
                              HayPieza => "HayVACSOP",
                              Pieza_Empaquetada => "VACSOPEnEMB");
   END_IF;
END_REGION

REGION Network 6: Maquina embalaje
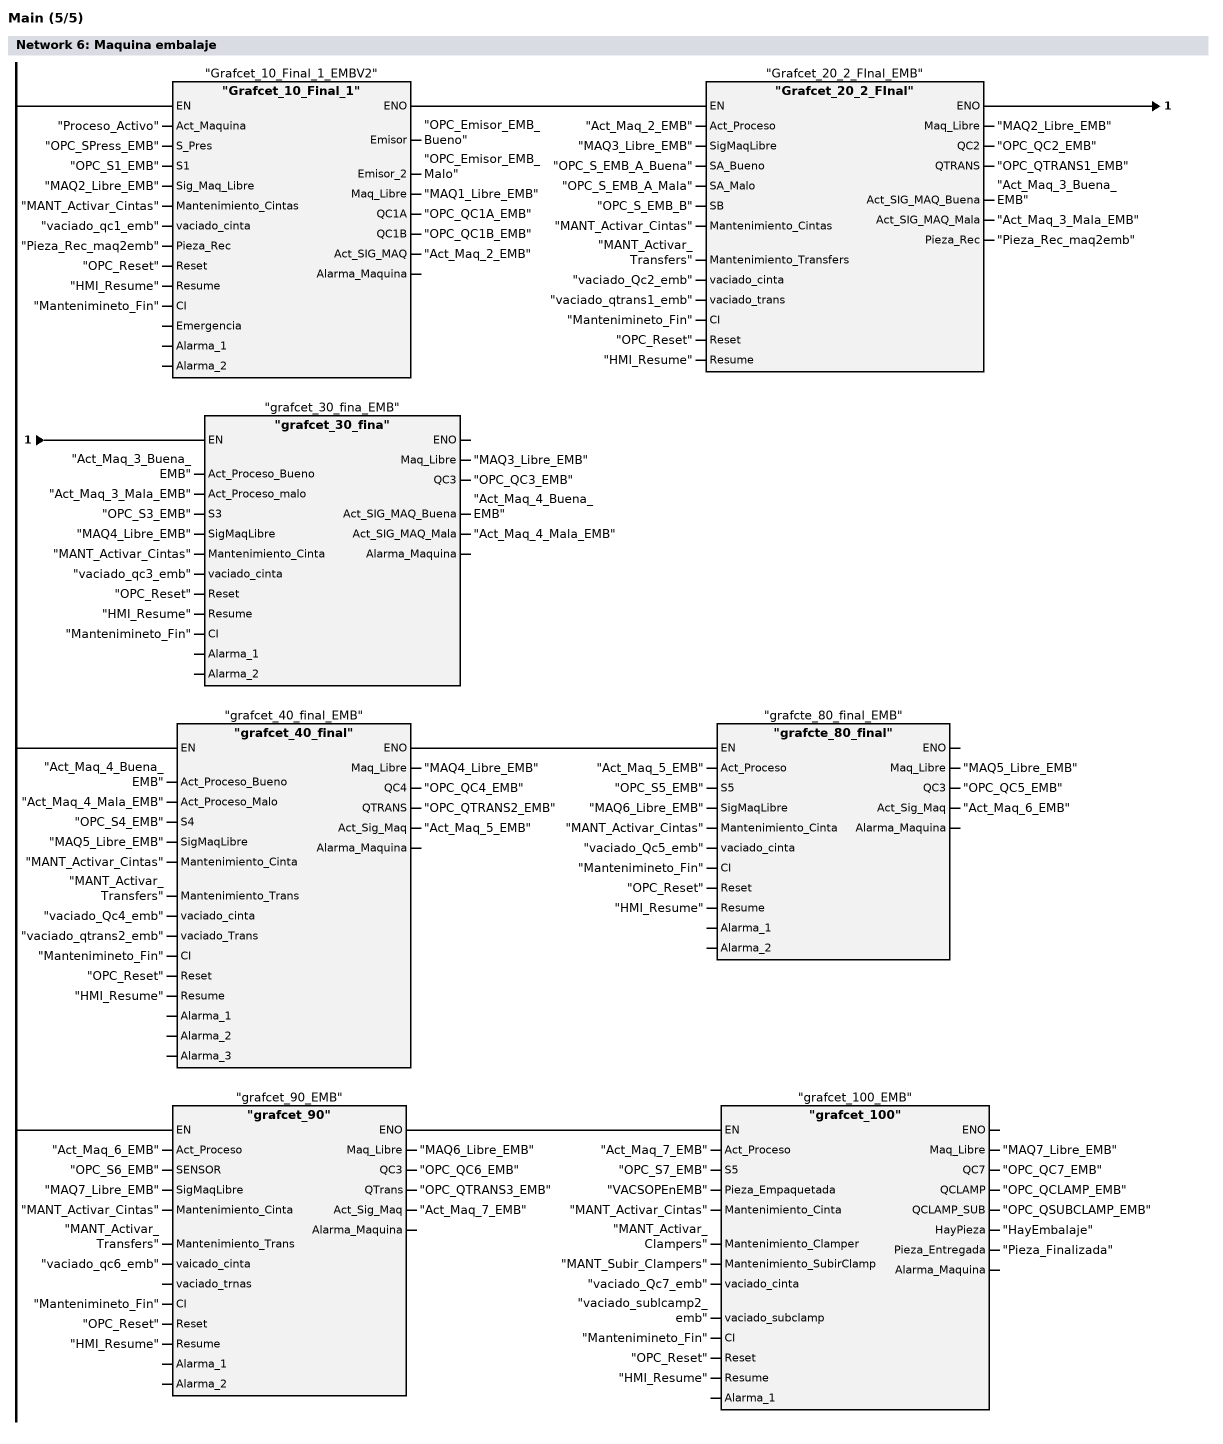
   RUNG wire#powerrail
      "Grafcet_10_Final_1_EMBV2"(Act_Maquina := "Proceso_Activo", S_Pres := "OPC_SPress_EMB", S1 := "OPC_S1_EMB", Sig_Maq_Libre := "MAQ2_Libre_EMB", Mantenimiento_Cintas := "MANT_Activar_Cintas", vaciado_cinta := "vaciado_qc1_emb", Pieza_Rec := "Pieza_Rec_maq2emb", Reset := "OPC_Reset", Resume := "HMI_Resume", CI := "Mantenimineto_Fin", Emergencia :=, Alarma_1 :=, Alarma_2 :=, Emisor => "OPC_Emisor_EMB_Bueno", Emisor_2 => "OPC_Emisor_EMB_Malo", Maq_Libre => "MAQ1_Libre_EMB", QC1A => "OPC_QC1A_EMB", QC1B => "OPC_QC1B_EMB", Act_SIG_MAQ => "Act_Maq_2_EMB", Alarma_Maquina =>)
      "Grafcet_20_2_FInal_EMB"(Act_Proceso := "Act_Maq_2_EMB", SigMaqLibre := "MAQ3_Libre_EMB", SA_Bueno := "OPC_S_EMB_A_Buena", SA_Malo := "OPC_S_EMB_A_Mala", SB := "OPC_S_EMB_B", Mantenimiento_Cintas := "MANT_Activar_Cintas", Mantenimiento_Transfers := "MANT_Activar_Transfers", vaciado_cinta := "vaciado_Qc2_emb", vaciado_trans := "vaciado_qtrans1_emb", CI := "Mantenimineto_Fin", Reset := "OPC_Reset", Resume := "HMI_Resume", Maq_Libre => "MAQ2_Libre_EMB", QC2 => "OPC_QC2_EMB", QTRANS => "OPC_QTRANS1_EMB", Act_SIG_MAQ_Buena => "Act_Maq_3_Buena_EMB", Act_SIG_MAQ_Mala => "Act_Maq_3_Mala_EMB", Pieza_Rec => "Pieza_Rec_maq2emb")
      "grafcet_30_fina_EMB"(Act_Proceso_Bueno := "Act_Maq_3_Buena_EMB", Act_Proceso_malo := "Act_Maq_3_Mala_EMB", S3 := "OPC_S3_EMB", SigMaqLibre := "MAQ4_Libre_EMB", Mantenimiento_Cinta := "MANT_Activar_Cintas", vaciado_cinta := "vaciado_qc3_emb", Reset := "OPC_Reset", Resume := "HMI_Resume", CI := "Mantenimineto_Fin", Alarma_1 :=, Alarma_2 :=, Maq_Libre => "MAQ3_Libre_EMB", QC3 => "OPC_QC3_EMB", Act_SIG_MAQ_Buena => "Act_Maq_4_Buena_EMB", Act_SIG_MAQ_Mala => "Act_Maq_4_Mala_EMB", Alarma_Maquina =>)
   END_RUNG
   RUNG wire#powerrail
      "grafcet_40_final_EMB"(Act_Proceso_Bueno := "Act_Maq_4_Buena_EMB", Act_Proceso_Malo := "Act_Maq_4_Mala_EMB", S4 := "OPC_S4_EMB", SigMaqLibre := "MAQ5_Libre_EMB", Mantenimiento_Cinta := "MANT_Activar_Cintas", Mantenimiento_Trans := "MANT_Activar_Transfers", vaciado_cinta := "vaciado_Qc4_emb", vaciado_Trans := "vaciado_qtrans2_emb", CI := "Mantenimineto_Fin", Reset := "OPC_Reset", Resume := "HMI_Resume", Alarma_1 :=, Alarma_2 :=, Alarma_3 :=, Maq_Libre => "MAQ4_Libre_EMB", QC4 => "OPC_QC4_EMB", QTRANS => "OPC_QTRANS2_EMB", Act_Sig_Maq => "Act_Maq_5_EMB", Alarma_Maquina =>)
      "grafcte_80_final_EMB"(Act_Proceso := "Act_Maq_5_EMB", S5 := "OPC_S5_EMB", SigMaqLibre := "MAQ6_Libre_EMB", Mantenimiento_Cinta := "MANT_Activar_Cintas", vaciado_cinta := "vaciado_Qc5_emb", CI := "Mantenimineto_Fin", Reset := "OPC_Reset", Resume := "HMI_Resume", Alarma_1 :=, Alarma_2 :=, Maq_Libre => "MAQ5_Libre_EMB", QC3 => "OPC_QC5_EMB", Act_Sig_Maq => "Act_Maq_6_EMB", Alarma_Maquina =>)
   END_RUNG
   RUNG wire#powerrail
      "grafcet_90_EMB"(Act_Proceso := "Act_Maq_6_EMB", SENSOR := "OPC_S6_EMB", SigMaqLibre := "MAQ7_Libre_EMB", Mantenimiento_Cinta := "MANT_Activar_Cintas", Mantenimiento_Trans := "MANT_Activar_Transfers", vaicado_cinta := "vaciado_qc6_emb", vaciado_trnas :=, CI := "Mantenimineto_Fin", Reset := "OPC_Reset", Resume := "HMI_Resume", Alarma_1 :=, Alarma_2 :=, Maq_Libre => "MAQ6_Libre_EMB", QC3 => "OPC_QC6_EMB", QTrans => "OPC_QTRANS3_EMB", Act_Sig_Maq => "Act_Maq_7_EMB", Alarma_Maquina =>)
      "grafcet_100_EMB"(Act_Proceso := "Act_Maq_7_EMB", S5 := "OPC_S7_EMB", Pieza_Empaquetada := "VACSOPEnEMB", Mantenimiento_Cinta := "MANT_Activar_Cintas", Mantenimiento_Clamper := "MANT_Activar_Clampers", Mantenimiento_SubirClamp := "MANT_Subir_Clampers", vaciado_cinta := "vaciado_Qc7_emb", vaciado_subclamp := "vaciado_sublcamp2_emb", CI := "Mantenimineto_Fin", Reset := "OPC_Reset", Resume := "HMI_Resume", Alarma_1 :=, Maq_Libre => "MAQ7_Libre_EMB", QC7 => "OPC_QC7_EMB", QCLAMP => "OPC_QCLAMP_EMB", QCLAMP_SUB => "OPC_QSUBCLAMP_EMB", HayPieza => "HayEmbalaje", Pieza_Entregada => "Pieza_Finalizada", Alarma_Maquina =>)
   END_RUNG
   // the same network as SCL:
   "Grafcet_10_Final_1_EMBV2"(Act_Maquina := "Proceso_Activo",   // "Grafcet_10_Final_1"
                           S_Pres := "OPC_SPress_EMB",
                           S1 := "OPC_S1_EMB",
                           Sig_Maq_Libre := "MAQ2_Libre_EMB",
                           Mantenimiento_Cintas := "MANT_Activar_Cintas",
                           vaciado_cinta := "vaciado_qc1_emb",
                           Pieza_Rec := "Pieza_Rec_maq2emb",
                           Reset := "OPC_Reset",
                           Resume := "HMI_Resume",
                           CI := "Mantenimineto_Fin",
                           Emisor => "OPC_Emisor_EMB_Bueno",
                           Emisor_2 => "OPC_Emisor_EMB_Malo",
                           Maq_Libre => "MAQ1_Libre_EMB",
                           QC1A => "OPC_QC1A_EMB",
                           QC1B => "OPC_QC1B_EMB",
                           Act_SIG_MAQ => "Act_Maq_2_EMB",
                           ENO => #_w1);
   "Grafcet_20_2_FInal_EMB"(EN := #_w1,   // "Grafcet_20_2_FInal"
                           Act_Proceso := "Act_Maq_2_EMB",
                           SigMaqLibre := "MAQ3_Libre_EMB",
                           SA_Bueno := "OPC_S_EMB_A_Buena",
                           SA_Malo := "OPC_S_EMB_A_Mala",
                           SB := "OPC_S_EMB_B",
                           Mantenimiento_Cintas := "MANT_Activar_Cintas",
                           Mantenimiento_Transfers := "MANT_Activar_Transfers",
                           vaciado_cinta := "vaciado_Qc2_emb",
                           vaciado_trans := "vaciado_qtrans1_emb",
                           CI := "Mantenimineto_Fin",
                           Reset := "OPC_Reset",
                           Resume := "HMI_Resume",
                           Maq_Libre => "MAQ2_Libre_EMB",
                           QC2 => "OPC_QC2_EMB",
                           QTRANS => "OPC_QTRANS1_EMB",
                           Act_SIG_MAQ_Buena => "Act_Maq_3_Buena_EMB",
                           Act_SIG_MAQ_Mala => "Act_Maq_3_Mala_EMB",
                           Pieza_Rec => "Pieza_Rec_maq2emb",
                           ENO => #_w2);
   IF #_w2 THEN
       "grafcet_30_fina_EMB"(Act_Proceso_Bueno := "Act_Maq_3_Buena_EMB",   // "grafcet_30_fina"
                             Act_Proceso_malo := "Act_Maq_3_Mala_EMB",
                             S3 := "OPC_S3_EMB",
                             SigMaqLibre := "MAQ4_Libre_EMB",
                             Mantenimiento_Cinta := "MANT_Activar_Cintas",
                             vaciado_cinta := "vaciado_qc3_emb",
                             Reset := "OPC_Reset",
                             Resume := "HMI_Resume",
                             CI := "Mantenimineto_Fin",
                             Maq_Libre => "MAQ3_Libre_EMB",
                             QC3 => "OPC_QC3_EMB",
                             Act_SIG_MAQ_Buena => "Act_Maq_4_Buena_EMB",
                             Act_SIG_MAQ_Mala => "Act_Maq_4_Mala_EMB");
   END_IF;
   "grafcet_40_final_EMB"(Act_Proceso_Bueno := "Act_Maq_4_Buena_EMB",   // "grafcet_40_final"
                          Act_Proceso_Malo := "Act_Maq_4_Mala_EMB",
                          S4 := "OPC_S4_EMB",
                          SigMaqLibre := "MAQ5_Libre_EMB",
                          Mantenimiento_Cinta := "MANT_Activar_Cintas",
                          Mantenimiento_Trans := "MANT_Activar_Transfers",
                          vaciado_cinta := "vaciado_Qc4_emb",
                          vaciado_Trans := "vaciado_qtrans2_emb",
                          CI := "Mantenimineto_Fin",
                          Reset := "OPC_Reset",
                          Resume := "HMI_Resume",
                          Maq_Libre => "MAQ4_Libre_EMB",
                          QC4 => "OPC_QC4_EMB",
                          QTRANS => "OPC_QTRANS2_EMB",
                          Act_Sig_Maq => "Act_Maq_5_EMB",
                          ENO => #_w3);
   IF #_w3 THEN
       "grafcte_80_final_EMB"(Act_Proceso := "Act_Maq_5_EMB",   // "grafcte_80_final"
                              S5 := "OPC_S5_EMB",
                              SigMaqLibre := "MAQ6_Libre_EMB",
                              Mantenimiento_Cinta := "MANT_Activar_Cintas",
                              vaciado_cinta := "vaciado_Qc5_emb",
                              CI := "Mantenimineto_Fin",
                              Reset := "OPC_Reset",
                              Resume := "HMI_Resume",
                              Maq_Libre => "MAQ5_Libre_EMB",
                              QC3 => "OPC_QC5_EMB",
                              Act_Sig_Maq => "Act_Maq_6_EMB");
   END_IF;
   "grafcet_90_EMB"(Act_Proceso := "Act_Maq_6_EMB",   // "grafcet_90"
                    SENSOR := "OPC_S6_EMB",
                    SigMaqLibre := "MAQ7_Libre_EMB",
                    Mantenimiento_Cinta := "MANT_Activar_Cintas",
                    Mantenimiento_Trans := "MANT_Activar_Transfers",
                    vaicado_cinta := "vaciado_qc6_emb",
                    CI := "Mantenimineto_Fin",
                    Reset := "OPC_Reset",
                    Resume := "HMI_Resume",
                    Maq_Libre => "MAQ6_Libre_EMB",
                    QC3 => "OPC_QC6_EMB",
                    QTrans => "OPC_QTRANS3_EMB",
                    Act_Sig_Maq => "Act_Maq_7_EMB",
                    ENO => #_w4);
   IF #_w4 THEN
       "grafcet_100_EMB"(Act_Proceso := "Act_Maq_7_EMB",   // "grafcet_100"
                         S5 := "OPC_S7_EMB",
                         Pieza_Empaquetada := "VACSOPEnEMB",
                         Mantenimiento_Cinta := "MANT_Activar_Cintas",
                         Mantenimiento_Clamper := "MANT_Activar_Clampers",
                         Mantenimiento_SubirClamp := "MANT_Subir_Clampers",
                         vaciado_cinta := "vaciado_Qc7_emb",
                         vaciado_subclamp := "vaciado_sublcamp2_emb",
                         CI := "Mantenimineto_Fin",
                         Reset := "OPC_Reset",
                         Resume := "HMI_Resume",
                         Maq_Libre => "MAQ7_Libre_EMB",
                         QC7 => "OPC_QC7_EMB",
                         QCLAMP => "OPC_QCLAMP_EMB",
                         QCLAMP_SUB => "OPC_QSUBCLAMP_EMB",
                         HayPieza => "HayEmbalaje",
                         Pieza_Entregada => "Pieza_Finalizada");
   END_IF;
END_REGION
END_ORGANIZATION_BLOCK

(* ===== HMI "HMI_RT_2" =====
system functions are stored by id; their names below are inferred from use
connection "HMI_Connection_1": ETHERNET, S7_1500_OMS

HMI tags "Default tag table"
   "HMI_Marcha" : Bool = PLC HMI_Marcha AT %M10.6, 1 s

discrete alarms
   1: 'MAQ 1 Vacuna - Alarma', class Errors
   2: 'MAQ 2 Vacuna - Alarma', class Errors bit 0
   3: 'MAQ 3 Vacuna - Alarma', class Errors bit 0
   4: 'MAQ 4 Vacuna - Alarma', class Errors bit 0
   5: 'MAQ 5 Vacuna - Alarma', class Errors bit 0
   6: 'MAQ 1 Soporte - Alarma', class Errors
   7: 'MAQ 2 Soporte - Alarma', class Errors bit 0
   8: 'MAQ 3 Soporte - Alarma', class Errors bit 0
   9: 'MAQ 4 Soporte - Alarma', class Errors bit 0
   10: 'MAQ 5 Soporte - Alarma', class Errors bit 0
   11: 'MAQ 6 Soporte - Alarma', class Errors bit 0
   12: 'MAQ 1 Embalaje - Alarma', class Errors
   13: 'MAQ 2 Embalaje - Alarma', class Errors bit 0
   14: 'MAQ 3 Embalaje - Alarma', class Errors bit 0
   15: 'MAQ 4 Embalaje - Alarma', class Errors bit 0
   16: 'MAQ 5 Embalaje - Alarma', class Errors bit 0
   17: 'MAQ 6 Embalaje - Alarma', class Errors bit 0
   18: 'MAQ 7 Embalaje - Alarma', class Errors bit 0

screen "MAIN" 1366x768
   GraphicView "Graphic view_1" at 0,0 size 1364x766; Picture "Graphic_1"
   Button "Button_1" at 1168,651 size 170x107; TextOff 'Modo Principal'
   Button "Button_2" at 12,23 size 294x158; TextOff 'Marcha'
      on Release: ResetBit("HMI_Marcha")
      on Press: SetBit("HMI_Marcha")
   Button "Button_3" at 15,197 size 294x158; TextOff 'Paro'
   Button "Button_4" at 15,372 size 294x158; TextOff 'RESUME'
   Button "Button_5" at 382,154 size 126x75; TextOff 'Text'
      on Press: ActivateScreen("Alarmas", 0)

screen "Alarmas" 1366x768
   AlarmView "Alarm view_1" at 97,69 size 1156x464
   Button "Button_1" at 444,556 size 164x88; TextOff 'RESET'
   Button "Button_2" at 672,556 size 164x88; TextOff 'RESUME'
   TextField "Text field_1" at 512,26 size 412x43; Text 'REGISTRO DE ALARMAS'
   Button "Button_3" at 72,688 size 156x62; TextOff 'VOLVER'
      on Press: function_efd93a16()
*)